# B&R Automation Studio project 305841_E00002_AM_0 (part 14)

#### ActionMotionFbs.st
```iecst
(********************************************************************
 * COPYRIGHT -- General Atomics
 ********************************************************************
 * Program: AxisStateMachine
 * File: ActionMoveVel.st
 * Author: Administrator
 * Created: January 22, 2014
 ********************************************************************
 * Implementation of program AxisStateMachine
 ********************************************************************)

ACTION ActionCallMotionFunctions:
  ActionMpAxisBasic;
  ActionCamInOut;
  ActionGearInOut;
  ActionOffsetShift;
  ActionPhaseShift;
END_ACTION

ACTION ActionMpAxisBasic:
  // 1) Range checks position, velocity, accel & Decel
  // 2) Packs the sMot_MoveParameters into a local axisBasicParamsStructure
  // 3) Detects parameter changes and manages the Update and UpdateDone bits
  // 4) Sets the fb command bits based on the axis sMot_AxisCommands structure
  // 5) Runs the fbMpAxisBasic funciton block
  // 6) Updates the axis structure with the status and axis info coming back from the fb

  // Make sure min/max values are not exceeded for position, velocity, accel, and decel.
  // Clamp if necessary

  // Position
  IF ax.MoveParameters.Position >  axPositionLimits.PositionLimitPos THEN
    ax.MoveParameters.Position :=  axPositionLimits.PositionLimitPos;
  END_IF;
  IF ax.MoveParameters.Position <  axPositionLimits.PositionLimitNeg THEN
    ax.MoveParameters.Position :=  axPositionLimits.PositionLimitNeg;
  END_IF;

  // Velocity
  IF ax.MoveParameters.Velocity > ax.MoveParameters.VelocityMax THEN
    ax.MoveParameters.Velocity := ax.MoveParameters.VelocityMax;
  END_IF;
  IF ax.MoveParameters.Velocity < ax.MoveParameters.VelocityMin THEN
    ax.MoveParameters.Velocity := ax.MoveParameters.VelocityMin;
  END_IF;

  // Accel and decel
  IF ax.MoveParameters.Acceleration > ax.MoveParameters.AccelMax THEN
    ax.MoveParameters.Acceleration := ax.MoveParameters.AccelMax;
  END_IF;
  IF ax.MoveParameters.Acceleration < ax.MoveParameters.AccelMin THEN
    ax.MoveParameters.Acceleration := ax.MoveParameters.AccelMin;
  END_IF;

  IF ax.MoveParameters.Deceleration > ax.MoveParameters.DecelMax THEN
    ax.MoveParameters.Deceleration := ax.MoveParameters.DecelMax;
  END_IF;
  IF ax.MoveParameters.Deceleration < ax.MoveParameters.DecelMin THEN
    ax.MoveParameters.Deceleration := ax.MoveParameters.DecelMin;
  END_IF;

  // The execution behavior is determined by the inputs set elsewhere
  // in particular the sMot_AxisCommands XxxxCmd bits,
  // and the values in sMot_MoveParameters structure

  // Axis reference set in init routine

  // Only enable the fb if the axis is not set to be ignored
  // TODO: Different check needed? Not sure how to tell if an axis reference is not set
  // It would be nice to check ax.fbMpAxisBasic.MpLink <> 0 for example, but this is a structure not an address
  IF NOT ax.Ignore AND ax.AxisNo <> 0 THEN
    ax.fbMpAxisBasic.Enable := TRUE;
  ELSE
    ax.fbMpAxisBasic.Enable := FALSE;
  END_IF;

  // Load the parameters from the sMot_MoveParameter structure into
  // local structure variables used for the fb
  fctPackMpAxisBasicParams(_I_UdtParams:= ADR(ax.MoveParameters), _IO_MpParams := axisBasicParams);

  // To allow move parameter changes to take effect without having to stop,
  // detect a difference between the desired parameters and the previous values.
  // If they are different, then set the update bit until the UpdateDone bit is set.
  // NOTE: This fb manages the ax.fbMpAxisCoupling.Update request and monitors the .UpdateDone bit
  // Use the .UpdateCouplingParams bit in the command structure if the application needs to control
  // when to trigger the update. If parameters need to be set in possibly different areas of the software,
  // and all the updates should take place at once, the update fb is called conditionally. The
  // checked bit can be set high so it is called all the time if the checked bit is not managed.
  ax.Commands.UpdateMoveParams:= TRUE;
  IF ax.Commands.UpdateMoveParams THEN
    ax.fbUpdateBFbParams(_IO_MpParams := axisBasicParams);
    ax.Commands.UpdateMoveParams := FALSE;
  END_IF;

  // TODO: Enforce move permissives

  // Use the commands from the axis structue
  ax.fbMpAxisBasic.ErrorReset := ax.Commands.DriveResetCmd;
  ax.fbMpAxisBasic.Power := ax.Commands.EnableCmd;
  ax.fbMpAxisBasic.Home := ax.Commands.HomeCmd;
  // There is no specific jog cmd. Use Move Velocity instead.
  ax.fbMpAxisBasic.MoveVelocity := ax.Commands.MoveVelocityCmd OR ax.Commands.MoveJogCmd;
  ax.fbMpAxisBasic.MoveAbsolute := ax.Commands.MoveAbsoluteCmd;
  ax.fbMpAxisBasic.MoveAdditive := ax.Commands.MoveRelativeCmd;
  ax.fbMpAxisBasic.Stop := ax.Commands.StopCmd;
  ax.fbMpAxisBasic.JogPositive := ax.Commands.MoveJogPositiveCmd;
  ax.fbMpAxisBasic.JogNegative := ax.Commands.MoveJogNegativeCmd;
  ax.fbMpAxisBasic.LimitLoad := ax.MoveParameters.EnableTorqueLimit;
  ax.fbMpAxisBasic.ReleaseBrake := ax.Commands.ReleaseBrakeCmd;
  ax.fbMpAxisBasic.AutoTune := FALSE; // TODO
  ax.fbMpAxisBasic.Simulate := FALSE; // TODO

  // Call the fb
  ax.fbMpAxisBasic();

  // Update the axis status structure
  ax.Status.Position := ax.fbMpAxisBasic.Position;
  ax.Status.Velocity := ax.fbMpAxisBasic.Velocity;
  ax.Status.IsPoweredOn := ax.fbMpAxisBasic.PowerOn;
  ax.Status.IsHomed := ax.fbMpAxisBasic.IsHomed;
  ax.Status.IsInVelocity := ax.fbMpAxisBasic.InVelocity;
  ax.Status.IsInPosition := ax.fbMpAxisBasic.InPosition;
  ax.Status.IsMoveActive := ax.fbMpAxisBasic.MoveActive;
  ax.Status.IsMoveDone := ax.fbMpAxisBasic.MoveDone;
  ax.Status.IsStopped := ax.fbMpAxisBasic.Stopped;
  ax.Status.IsTorqueLimitReady := ax.fbMpAxisBasic.LimitLoadReady;
  ax.Status.IsBrakeManuallyReleased := ax.fbMpAxisBasic.BrakeReleased;

  // Now load the sMot_AxisStatus structure with the data returned from the fb
  fctGetMpAxisInfo(_I_MpInfo := ADR(ax.fbMpAxisBasic.Info), _IO_UdtStatus := ax.Status);

  // Calculate special (algorithmic) positions
  CalcSpecialPositions;

  // Now that the status of this axis is known, copy it to the other axes slave status
  // area if this axis is specified as a slave.
  CopySlaveStatusToMaster;

END_ACTION

ACTION ActionCamInOut:
  // Execute the cam in or cam out fbs based on the CamIn/Out requests
  // The fbs are edge triggered, and the requests are cleared once serviced.
  // If the caming params change, another request must be made.
  // TODO: Is cam out and another cam in needed if params change?

  // Only execute the cam in fb if the axis number has been set,
  // the slave axis number has been set, and neither is set to be ignored,
  // and it is requested.
  IF ax.Ignore OR ax.AxisNo = AD_UNKNOWN OR
       ax.CouplingParameters.SlaveAxisNo = AD_UNKNOWN OR
       axes[ax.CouplingParameters.SlaveAxisNo].Ignore THEN
    // slave or master should be ignored
    // keep the requests and executes low
    ax.CouplingParameters.CamInReq := FALSE;
    ax.CouplingParameters.CamOutReq := FALSE;
    ax.fbCamIn.Execute := FALSE;
    ax.fbCamOut.Execute := FALSE;
  ELSIF ax.CouplingParameters.CamInReq THEN
    // CamIn request is made.
    // Clear the req so a future rising edge can be seen
    ax.CouplingParameters.CamInReq := FALSE;
    // Make sure the CamOut req and execute is clear
    ax.CouplingParameters.CamOutReq := FALSE;
    ax.fbCamOut.Execute := FALSE;
    // Load the cam in params, then set the execute input (edge triggered fb)
    ax.fbCamIn.MasterOffset := ax.CouplingParameters.CamMasterOffset;
    ax.fbCamIn.SlaveOffset := ax.CouplingParameters.CamSlaveOffset;
    ax.fbCamIn.MasterScaling := ax.CouplingParameters.CamScalingMaster;
    ax.fbCamIn.SlaveScaling := ax.CouplingParameters.CamScalingSlave;
    ax.fbCamIn.StartMode := ax.CouplingParameters.CamStartMode;
    ax.fbCamIn.MasterValueSource := ax.CouplingParameters.CamMasterValueSource;
    ax.fbCamIn.CamID := ax.CouplingParameters.CamId;
    ax.fbCamIn.BufferMode := ax.CouplingParameters.CamBufferMode; // only mcAborting currently supported
    ax.fbCamIn.AdvancedParameters.Periodic := ax.CouplingParameters.CamIsPeriodic;
    ax.fbCamIn.AdvancedParameters.Velocity := 0.0; // disable, use (slave?) axis max vel
    ax.fbCamIn.AdvancedParameters.Acceleration := 0.0; // disable, use (slave?) axis max accel
    ax.fbCamIn.AdvancedParameters.Deceleration := 0.0; // disable, use (slave?) axis max decel
    ax.fbCamIn.AdvancedParameters.Jerk := 0.0; // only non-zero if using McProfGen
    ax.fbCamIn.Execute := TRUE; // fb looks for a rising edge
  ELSIF ax.CouplingParameters.CamOutReq THEN
    // Clear the req so a future rising edge can be seen
    ax.CouplingParameters.CamOutReq := FALSE;
    // Make sure the GearIn req and execute is clear
    ax.CouplingParameters.CamInReq := FALSE;
    ax.fbCamIn.Execute := FALSE;
    // Load the cam out params, then set the execute input (edge triggered fb)
    ax.fbCamOut.Jerk := 0.0; // only non-zero if using McProfGen
    ax.fbCamOut.Execute := TRUE;
  END_IF;

  // Call the cam in and cam out fbs.
  ax.fbCamIn();
  ax.fbCamOut();
  // Clear the exuecute bits. The fbs are edge triggerd, and would have been seen by the above call.
  ax.fbCamIn.Execute := FALSE;
  ax.fbCamOut.Execute := FALSE;

  // Update the axis status structure
  IF ax.fbCamIn.Active AND NOT ax.fbCamIn.Error THEN
    ax.Status.IsCamInSync := ax.fbCamIn.InSync;
    ax.Status.IsCamEndOfProfile := ax.fbCamIn.EndOfProfile;
    ax.Status.CamStatus := ax.fbCamIn.Status;
  ELSE
    ax.Status.IsCamInSync := FALSE;
    ax.Status.IsCamEndOfProfile := FALSE;
    ax.Status.CamStatus := mcCAM_STATUS_PREPARING_MOVE; // 0 value, but don't have a good choice for "not active
  END_IF;

END_ACTION

ACTION ActionGearInOut:
  // Execute the gear in or gear out fbs based on the GearIn/Out requests
  // The fbs are edge triggered, and the requests are cleared once serviced.
  // If the gearing params change, another request must be made.

  // Only execute the gear in fb if the axis number has been set,
  // the slave axis number has been set, and neither is set to be ignored,
  // and it is requested.
  IF ax.Ignore OR ax.AxisNo = AD_UNKNOWN OR
       ax.CouplingParameters.SlaveAxisNo = AD_UNKNOWN OR
       axes[ax.CouplingParameters.SlaveAxisNo].Ignore THEN
    // slave or master should be ignored
    // keep the requests and executes low
    ax.CouplingParameters.GearInReq := FALSE;
    ax.CouplingParameters.GearOutReq := FALSE;
    ax.fbGearIn.Execute := FALSE;
    ax.fbGearOut.Execute := FALSE;
  ELSIF ax.CouplingParameters.GearInReq THEN
    // GearIn request is made.
    // Clear the req so a future rising edge can be seen
    ax.CouplingParameters.GearInReq := FALSE;
    // Make sure the GearOut req and execute is clear
    ax.CouplingParameters.GearOutReq := FALSE;
    ax.fbGearOut.Execute := FALSE;
    // Load the gear in params, then set the execute input (edge triggered fb)
    ax.fbGearIn.RatioNumerator := ax.CouplingParameters.GearInRatioNumerator;
    ax.fbGearIn.RatioDenominator := ax.CouplingParameters.GearInRatioDenominator;
    ax.fbGearIn.MasterValueSource := ax.CouplingParameters.GearInMasterValueSource;
    ax.fbGearIn.Acceleration := ax.CouplingParameters.ShiftAccelerationMax;
    ax.fbGearIn.Deceleration := ax.CouplingParameters.ShiftDecelerationMax;
    ax.fbGearIn.Jerk := ax.CouplingParameters.ShiftJerk; // only non-zero if using McProfGen
    ax.fbGearIn.BufferMode := ax.CouplingParameters.GearInBufferMode; // onlly mcAborting currently supported
    ax.fbGearIn.AdvancedParameters.MasterMaxVelocity := ax.CouplingParameters.ShiftProfileBaseMaxVelocity;
    ax.fbGearIn.Execute := TRUE; // fb looks for a rising edge
  ELSIF ax.CouplingParameters.GearOutReq THEN
    // Clear the req so a future rising edge can be seen
    ax.CouplingParameters.GearOutReq := FALSE;
    // Make sure the GearIn req and execute is clear
    ax.CouplingParameters.GearInReq := FALSE;
    ax.fbGearIn.Execute := FALSE;
    // Load the gear out params, then set the execute input (edge triggered fb)
    ax.fbGearOut.Jerk := 0.0; // only non-zero if using McProfGen
    ax.fbGearOut.Execute := TRUE;
  END_IF;

  // Call the gear in and gear out fbs.
  ax.fbGearIn();
  ax.fbGearOut();
  // Clear the exuecute bits. The fbs are edge triggerd, and would have been seen by the above call.
  ax.fbGearIn.Execute := FALSE;
  ax.fbGearOut.Execute := FALSE;

  // Update the axis status structure.
  // Derrive InCompensation -- Active but not in sync
  IF ax.fbGearIn.Active AND NOT ax.fbGearIn.Error THEN
    // If gear in is active, it is either in sync or in compensation
    ax.Status.IsGearInSync := ax.fbGearIn.InGear;
    ax.Status.IsGearInCompensation := NOT ax.fbGearIn.InGear;
  ELSE
    ax.Status.IsGearInSync := FALSE;
    ax.Status.IsGearInCompensation := FALSE;
  END_IF;

END_ACTION

ACTION ActionOffsetShift:
  // Execute the offset shift fb based on the offset shift request.
  // The fb is edge triggered, and the request is cleared once serviced.
  // If the offset params change, another request must be made.

  // Only execute the offset shift fb if the axis number has been set,
  // the slave axis number has been set, and neither is set to be ignored,
  // and it is requested.
  IF ax.Ignore OR ax.AxisNo = AD_UNKNOWN OR
       ax.CouplingParameters.SlaveAxisNo = AD_UNKNOWN OR
       axes[ax.CouplingParameters.SlaveAxisNo].Ignore THEN
    // slave or master should be ignored
    // keep the request and enable low
    ax.CouplingParameters.OffsetShiftReq := FALSE;
    ax.fbOffsetShift.Enable := FALSE;
    ax.fbOffsetShift.StartShift := FALSE;
  ELSE
    ax.fbOffsetShift.Enable := TRUE;
  END_IF;

  // Enable input and ignore considered above. If req is high,
  // it can be acted upon.
  IF ax.CouplingParameters.OffsetShiftReq THEN
    // Offset Shift request is made.
    // Clear the req so a future rising edge can be seen
    ax.CouplingParameters.OffsetShiftReq := FALSE;
    // Load the offset shift params, then set the start shift input (edge sensitive input)
    ax.fbOffsetShift.OffsetShift := ax.CouplingParameters.Shift;
    ax.fbOffsetShift.Velocity := ax.CouplingParameters.ShiftVelocityMax;
    ax.fbOffsetShift.Acceleration := ax.CouplingParameters.ShiftAccelerationMax;
    ax.fbOffsetShift.AdvancedParameters.ShiftMode := ax.CouplingParameters.ShiftMode;
    ax.fbOffsetShift.AdvancedParameters.ProfileBase := ax.CouplingParameters.ShiftProfileBase;
    ax.fbOffsetShift.AdvancedParameters.ProfileBaseMaxVelocity := ax.CouplingParameters.ShiftProfileBaseMaxVelocity;
    ax.fbOffsetShift.AdvancedParameters.DistanceParameters.ProfileDistance := ax.CouplingParameters.ShiftProfileDistance;
    ax.fbOffsetShift.AdvancedParameters.ZoneParameters.StartPosition := ax.CouplingParameters.ShiftZoneStartPosition;
    ax.fbOffsetShift.AdvancedParameters.ZoneParameters.EndPosition := ax.CouplingParameters.ShiftZoneEndPosition;
    ax.fbOffsetShift.AdvancedParameters.ZoneParameters.Period := ax.CouplingParameters.ShiftZonePeriod;
    ax.fbOffsetShift.AdvancedParameters.ShiftAlternativeValueSource := mcALT_VALUE_NOT_USED;
    ax.fbOffsetShift.StartShift := TRUE; // fb looks for a rising edge
  END_IF;

  // Call the offset shift fb.
  ax.fbOffsetShift();
  // Clear the start shift bit. The fb is edge triggerd, and it would have been seen by the above call.
  ax.fbOffsetShift.StartShift := FALSE; // fb looks for a rising edge

  // Update the axis status structure as long as status is valid and there is no error.
  // Otherwise, clear the values
  IF ax.fbOffsetShift.Valid AND NOT ax.fbOffsetShift.Error THEN
    ax.Status.IsCoordOffsetShiftAttained := ax.fbOffsetShift.ShiftAttained;
    ax.Status.IsCoordOffsetShiftStarted := ax.fbOffsetShift.ShiftStarted;
    ax.Status.CoordActualOffsetShift := ax.fbOffsetShift.ActualOffsetShift;
  ELSE
    ax.Status.IsCoordOffsetShiftAttained := FALSE;
    ax.Status.IsCoordOffsetShiftStarted := FALSE;
    ax.Status.CoordActualOffsetShift := 0.0;
  END_IF;

END_ACTION

ACTION ActionPhaseShift:
  // Execute the phase shift fb based on the phase shift request.
  // The fb is edge triggered, and the request is cleared once serviced.
  // If the phase params change, another request must be made.
  // TODO: Verify operation/behavior when changing params

  // Only execute the phase shift fb if the axis number has been set,
  // the slave axis number has been set, and neither is set to be ignored,
  // and it is requested.
  IF ax.Ignore OR ax.AxisNo = AD_UNKNOWN OR
       ax.CouplingParameters.SlaveAxisNo = AD_UNKNOWN OR
       axes[ax.CouplingParameters.SlaveAxisNo].Ignore THEN
    // slave or master should be ignored
    // keep the request and enable low
    ax.CouplingParameters.PhaseShiftReq := FALSE;
    ax.fbPhaseShift.Enable := FALSE;
    ax.fbPhaseShift.StartShift := FALSE;
  ELSE
    ax.fbPhaseShift.Enable := TRUE;
  END_IF;

  // Enable input and ignore considered above. If req is high,
  // it can be acted upon.
  IF ax.CouplingParameters.PhaseShiftReq THEN
    // Phase Shift request is made.
    // Clear the req so a future rising edge can be seen
    ax.CouplingParameters.PhaseShiftReq := FALSE;
    // Load the phase shift params, then set the start shift input (edge sensitive input)
    ax.fbPhaseShift.PhaseShift := ax.CouplingParameters.Shift;
    ax.fbPhaseShift.Velocity := ax.CouplingParameters.ShiftVelocityMax;
    ax.fbOffsetShift.Acceleration := ax.CouplingParameters.ShiftAccelerationMax;
    ax.fbOffsetShift.AdvancedParameters.ShiftMode := ax.CouplingParameters.ShiftMode;
    ax.fbOffsetShift.AdvancedParameters.ProfileBase := ax.CouplingParameters.ShiftProfileBase;
    ax.fbOffsetShift.AdvancedParameters.ProfileBaseMaxVelocity := ax.CouplingParameters.ShiftProfileBaseMaxVelocity;
    ax.fbOffsetShift.AdvancedParameters.DistanceParameters.ProfileDistance := ax.CouplingParameters.ShiftProfileDistance;
    ax.fbOffsetShift.AdvancedParameters.ZoneParameters.StartPosition := ax.CouplingParameters.ShiftZoneStartPosition;
    ax.fbOffsetShift.AdvancedParameters.ZoneParameters.EndPosition := ax.CouplingParameters.ShiftZoneEndPosition;
    ax.fbOffsetShift.AdvancedParameters.ZoneParameters.Period := ax.CouplingParameters.ShiftZonePeriod;
    ax.fbOffsetShift.AdvancedParameters.ShiftAlternativeValueSource := mcALT_VALUE_NOT_USED;
    ax.fbPhaseShift.StartShift := TRUE; // fb looks for a rising edge
  END_IF;

  // Call the phase shift fb.
  ax.fbPhaseShift();
  // Clear the start shift bit. The fb is edge triggerd, and it would have been seen by the above call.
  ax.fbPhaseShift.StartShift := FALSE; // fb looks for a rising edge

  // Update the axis status structure as long as status is valid and there is no error.
  // Otherwise, clear the values
  IF ax.fbPhaseShift.Valid AND NOT ax.fbPhaseShift.Error THEN
    ax.Status.IsCoordPhaseShiftAttained := ax.fbPhaseShift.ShiftAttained;
    ax.Status.IsCoordPhaseShiftStarted := ax.fbPhaseShift.ShiftStarted;
    ax.Status.CoordActualPhaseShift := ax.fbPhaseShift.ActualPhaseShift;
  ELSE
    ax.Status.IsCoordPhaseShiftAttained := FALSE;
    ax.Status.IsCoordPhaseShiftStarted := FALSE;
    ax.Status.CoordActualPhaseShift := 0.0;
  END_IF;

END_ACTION

ACTION CopySlaveStatusToMaster :
  // If this axis number is a slave to another axis, then copy this axis
  // status to the master axis structure. This is a convenience
  // so the HMI for example, only needs to look in one structure (the master) and
  // can access the slave status.

  // Loop thru the axes. If the axis of index has this axis specified as a slave axis,
  // copy this axis status to the axis of index slave status.
  // Axis 0 is a dummy axis, so it can be skipped.
  FOR axIdx := 1 TO AXIS_COUNT DO
    IF axes[axIdx].CouplingParameters.SlaveAxisNo = AXIS_NO THEN
      // This axis is a slave to the axis referenced by axIdx.
      // Copy this axis status to the indexed axis slave status
      fctCopyAxisStatus(_I_SrcStatus := ADR(ax.Status), _I_DestStatus := ADR(axes[axIdx].StatusSlave));
    END_IF;
  END_FOR;
END_ACTION
```

- ActionMotionFbs.st.bak (not shown)

#### AxSMInit.st
```iecst
PROGRAM _INIT
  // set ax pointer to the element of the global sMot_Axis array
  ax ACCESS ADR(axes[AXIS_NO]);

  // set the position limits to point to the global permanent variable
  axPositionLimits ACCESS ADR(gr_AxisPositionLimits[AXIS_NO]);

  // Set the axis number and clear the ignore bit
  ax.AxisNo:= AXIS_NO;

  // **** These settings need to be reviewed/set for each axis
  ax.CouplingParameters.SlaveAxisNo := DINT_TO_USINT(AD_UNKNOWN); // This axis will have slaves, but it changes during run-time
  ax.Ignore := FALSE;
  ax.isAxisEndless := TRUE;
  ax.isAxisVirtual := TRUE;
  ax.isAxisInverter := FALSE;

  // Point to the mappMotion axis, and a slave if there is one
  ax.AxisObj := gvAxHw; // mappMotion axis -- see mappMotion in cfg view
  ax.SlaveAxisObj := axDummySlave; // slave axis for the handwheel is dynamic

  // Set the restore pos check fb
  // ax.fbCheckRestorePos.Axis := ADR(ax.AxisObj);
  // ax.fbCheckRestorePos.DataAddress := ADR(gr_AxHwRestorePos); // Set this per axis

  // Load the min/max velocity and accel/decel from constants
  // Note: Moves not used for virtual axes, so values are not important
  ax.MoveParameters.AccelMin := 0.001; // TODO: Not sure of a good value, but it should not be zero.
  ax.MoveParameters.AccelMax:= 10.0;
  ax.MoveParameters.DecelMin := 0.001; // TODO:Not sure of a good value, but it should not be zero.
  ax.MoveParameters.DecelMax:= 10.0;
  ax.MoveParameters.VelocityMin := 0.000;
  ax.MoveParameters.VelocityMax := 01.0;

  // **** The settings below don't normally need to be altered

  // set the fb axis references
  ax.fbMpAxisBasic.MpLink := ADR(ax.AxisObj);
  ax.fbReadDrivePos.Axis:= ADR(ax.AxisObj);
  ax.fbGearIn.Master := ADR(ax.AxisObj);
  ax.fbGearIn.Slave := ADR(ax.SlaveAxisObj);
  ax.fbGearOut.Slave := ADR(ax.SlaveAxisObj);
  ax.fbOffsetShift.Slave := ADR(ax.SlaveAxisObj);
  ax.fbPhaseShift.Slave := ADR(ax.SlaveAxisObj);
  ax.fbCamIn.Master := ADR(ax.AxisObj);
  ax.fbCamIn.Slave := ADR(ax.SlaveAxisObj);
  ax.fbCamOut.Slave := ADR(ax.SlaveAxisObj);
  ax.fbUpdateBFbParams._I_Axis := ADR(ax);

  // Set fb reference to local variables
  ax.fbMpAxisBasic.Parameters := ADR(axisBasicParams);

  // Set previous values for motion parameters so changes can be detected
  ax.MoveParametersPrev := ax.MoveParameters;

  // Clear commands and requests
  fctClearMotionCommands(_I_CmdMask := MACM_NOMASK, _IO_Commands := ax.Commands);
  fctClearMotionRequests(_I_ReqMask := MACM_NOMASK, _IO_Commands := ax.Commands);

  // set the move not allowed flag
  ax.Commands.MoveNotAllowed:= TRUE;

  // Set the most primitive status. If the axis is valid, the
  // full status will be updated later once comms is established, and the drive status is updated via MpAxisBasic
  ax.Status.IsCommuncationReady := FALSE;
  ax.Status.IsReadyToPowerOn := FALSE;

END_PROGRAM
```

### Program Logical/PlcLogic/axCfVfd/axCfVfdSM

#### AxSM.var
```iecst
(********************************************************************
 * COPYRIGHT -- General Atomics
 ********************************************************************
 * Program: AFtInSM
 * File: AFtInSM.var
 * Author: Administrator
 * Created: July 16, 2014
 ********************************************************************
 * Local variables of program AFtInSM
 ********************************************************************)
VAR CONSTANT
  (* axis number is per eAXIS_DESIGNATION *)
  (*
    AD_UNKNOWN := 0,
    AD_SPINDLE := 1,
    AD_OUTER_ECCENTRIC := 2,
    AD_INNER_ECCENTRIC := 3,
    AD_Z := 4,
    derrived axes
    AD_X := 5,
    AD_Y := 6,
    virual axes
    AD_HANDWHEEL := 7
    AD_CF_VFD := 8
  *)

  (* same info but different data types for convenience *)
  AXIS_NO : USINT := AD_CF_VFD; (* USINT so it can be used as an array index *)
  AXIS_DESIGNATION : eAXIS_DESIGNATION := AD_CF_VFD;

  END_VAR

  VAR
  ax : REFERENCE TO sMot_Axis;
  axPositionLimits : REFERENCE TO sMot_PositionLimits;
  axIdx : DINT; (* axis index *)
  axDummySlave : McAxisType;
	(* local versions of motion param structures -- used to make setting advanced params easier *)
  axisBasicParams : MpAxisBasicParType;
  tmrStepTO : TON; (* Step TO timer *)
  reqMask : DINT := MACM_NOMASK; (* request mask *)
  cmdMask : DINT := MACM_NOMASK; (* command mask *)
  tmrDriveReset : TON; (* auto issue drive reset while invalid also used to force minimum time in error states *)
	tmrModeMismatch : TON; (* mode mismatch timer *)
	tmrHomeMinimum : TON; (* force Home cmd to be present before transitioning *)
END_VAR
```

#### ActionChkPermissives.st
```iecst
(********************************************************************
 * COPYRIGHT -- General Atomics
 ********************************************************************
 * Program: AxisStateMachine
 * File: ActionCheckPermissiveJog.st
 * Author: Administrator
 * Created: June 02, 2014
 ********************************************************************
 * Implementation of program AxisStateMachine
 ********************************************************************)

ACTION ActionChkPermissiveContinuous:
  // Permissive check for continuous moves -- jogs and velocity
  // These moves have an undefined length

  // NOTE THE MOVE NOT ALLOWED FLAG: This aciton will set this flag if it finds the move to be in violation.
  // It does not clear the flag, however, and this allows several check actions to be called in a chain. If
  // at the end of all the calls, the flag is set, then it is intended that the overall application logic should
  // not allow the move.

  (* ***** WARNING CAUTION ****
  These checks have only primitive checks for taking into account current velocicy, deceleration, and stopping distance.
  This means that the permissives will try to honor position limits, and try to keep from over-running a limit,
  but may overshoot if you run right up to a limit.

  The stopping distance is calculated from the velocity and decel value, which is mathmatically correct, but
  in practice, the velocity value is approximate since it is sampled at a relatively slow rate.
  ***************************** *)

  // Calculate the stopping Distance if the axis is not virtual
  // If the axis in not moving, assume the velocity parameter for a move.
  // If the axis is moving, used the reported velocity
  // Stopping distance = Vavg * t => V/2 * V/decel => V^2/2*decel
  IF NOT ax.isAxisVirtual THEN
    IF  ax.Status.PlcOpenState = mcAXIS_CONTINUOUS_MOTION OR // Will probably be continuous or synchronized because
        ax.Status.PlcOpenState = mcAXIS_DISCRETE_MOTION OR
        ax.Status.PlcOpenState = mcAXIS_SYNCHRONIZED_MOTION THEN
      // Axis is moving ... Use reported velocity
      // Prevent against divide by zero by assuming a value if decel is zero
      IF ax.MoveParameters.Deceleration = 0.0 THEN
        // No valid decel. Use min decel
        ax.MoveParameters.PermissiveCheck.EstStoppingDistance := (ax.Status.Velocity ** 2) / (2.0 * ax.MoveParameters.DecelMin);
      ELSE
        // We have a decel value, so use that
        ax.MoveParameters.PermissiveCheck.EstStoppingDistance := (ax.Status.Velocity ** 2) / (2.0 * ax.MoveParameters.Deceleration);
      END_IF;
    ELSE
      // Axis is stopped ... assume parameter velocity
      // Prevent against divide by zero by assuming a small value if decel is zero
      IF ax.MoveParameters.Deceleration = 0.0 THEN
        // No valid decel. Use min decel.
        ax.MoveParameters.PermissiveCheck.EstStoppingDistance := (ax.MoveParameters.Velocity ** 2) / (2.0 * ax.MoveParameters.DecelMin);
      ELSE
        // We have a decel value, so use that
        ax.MoveParameters.PermissiveCheck.EstStoppingDistance := (ax.MoveParameters.Velocity ** 2) / (2.0 * ax.MoveParameters.Deceleration);
      END_IF;
    END_IF;
  ELSE
    // virtual axis does not allow moves, so done not need stopping distance.
    ax.MoveParameters.PermissiveCheck.EstStoppingDistance := 0.0;
  END_IF;

  // Check the directional move permissives and then check the allowable position range

  // Initially clear the Check Failed flag.
  // This will get set if any check fails.
  // It will get checked at the end and will get used to control the
  // move not allowed bit. The move not allowed bit was not used directly in the
  // intermediate checks to avoid it transiting until all the logic was complete
  ax.MoveParameters.PermissiveCheck.CheckFailed:= FALSE;

  // positive move permissive
  IF ax.MoveParameters.Direction = mcDIR_POSITIVE  AND NOT ax.MoveParameters.PosMovePermissive THEN
    ax.MoveParameters.PermissiveCheck.PermissiveHaltPos:= TRUE;
    ax.MoveParameters.PermissiveCheck.CheckFailed:= TRUE;
  ELSE
    ax.MoveParameters.PermissiveCheck.PermissiveHaltPos:= FALSE;
  END_IF;

  // negative move permissive
  IF ax.MoveParameters.Direction = mcDIR_NEGATIVE AND NOT ax.MoveParameters.NegMovePermissive THEN
    ax.MoveParameters.PermissiveCheck.PermissiveHaltNeg:= TRUE;
    ax.MoveParameters.PermissiveCheck.CheckFailed:= TRUE;
  ELSE
    ax.MoveParameters.PermissiveCheck.PermissiveHaltNeg:= FALSE;
  END_IF;

  // If the check passed the above, and the axis is not endless, then check the position limits
  IF NOT ax.MoveParameters.PermissiveCheck.CheckFailed AND NOT ax.isAxisEndless THEN
    // positive position window
    IF ax.MoveParameters.Direction = mcDIR_POSITIVE  AND
      (ax.Status.Position >=  axPositionLimits.PositionLimitPos OR
      ax.Status.Position + ax.MoveParameters.PermissiveCheck.EstStoppingDistance >=  axPositionLimits.PositionLimitPos) THEN
      ax.MoveParameters.PermissiveCheck.RangeLimitPos:= TRUE;
      ax.MoveParameters.PermissiveCheck.CheckFailed:= TRUE;
    ELSE
      ax.MoveParameters.PermissiveCheck.RangeLimitPos:= FALSE;
    END_IF;

    // negative position window
    IF ax.MoveParameters.Direction = mcDIR_NEGATIVE AND
      (ax.Status.Position <=  axPositionLimits.PositionLimitNeg OR
      ax.Status.Position - ax.MoveParameters.PermissiveCheck.EstStoppingDistance <=  axPositionLimits.PositionLimitNeg) THEN
      ax.MoveParameters.PermissiveCheck.RangeLimitNeg:= TRUE;
      ax.MoveParameters.PermissiveCheck.CheckFailed:= TRUE;
    ELSE
      ax.MoveParameters.PermissiveCheck.RangeLimitNeg:= FALSE;
    END_IF;
  ELSIF ax.isAxisEndless THEN
    // Axis is endless, so it won't fail on position range... clear the bits
    ax.MoveParameters.PermissiveCheck.RangeLimitPos := FALSE;
    ax.MoveParameters.PermissiveCheck.RangeLimitNeg := FALSE;
  END_IF;

  // Set move not allowed bit depending on the check failed flag
  IF ax.MoveParameters.PermissiveCheck.CheckFailed THEN
    // at least 1 permissive failed, don't allow the move
    ax.Commands.MoveNotAllowed:= TRUE;
  END_IF;

END_ACTION

ACTION ActionChkPermissiveRel:
  // Check the directional move permissives and then check the allowable position range

  // NOTE THE MOVE NOT ALLOWED FLAG: This aciton will set this flag if it finds the move to be in violation.
  // It does not clear the flag, however, and this allows several check actions to be called in a chain. If
  // at the end of all the calls, the flag is set, then it is intended that the overall application logic should
  // not allow the move.

  // Initially clear the Check Failed flag.
  // This will get set if any check fails.
  // It will get checked at the end and will get used to control the
  // move not allowed bit. The move not allowed bit was not used directly in the
  // intermediate checks to avoid it transiting until all the logic was complete
  ax.MoveParameters.PermissiveCheck.CheckFailed:= FALSE;

  // positive move permissive
  // if distance is > 0, move is positive
  IF ax.MoveParameters.Distance > 0 AND NOT ax.MoveParameters.PosMovePermissive THEN
    ax.MoveParameters.PermissiveCheck.PermissiveHaltPos:= TRUE;
    ax.MoveParameters.PermissiveCheck.CheckFailed:= TRUE;
  ELSE
    ax.MoveParameters.PermissiveCheck.PermissiveHaltPos:= FALSE;
  END_IF;

  // negative move permissive
  // if distance is < 0, move is negative
  IF ax.MoveParameters.Distance < 0 AND NOT ax.MoveParameters.NegMovePermissive THEN
    ax.MoveParameters.PermissiveCheck.PermissiveHaltNeg:= TRUE;
    ax.MoveParameters.PermissiveCheck.CheckFailed:= TRUE;
  ELSE
    ax.MoveParameters.PermissiveCheck.PermissiveHaltNeg:= FALSE;
  END_IF;

  // If the check passed the above, and the axis is not endless, then check the position limits
  IF NOT ax.MoveParameters.PermissiveCheck.CheckFailed AND NOT ax.isAxisEndless THEN
    // positive position window -- if distance is > 0, move is positive
    IF ax.MoveParameters.Distance > 0.0 AND
      ax.MoveParameters.PermissiveCheck.StartPosition + ax.MoveParameters.Distance > axPositionLimits.PositionLimitPos THEN
      ax.MoveParameters.PermissiveCheck.RangeLimitPos:= TRUE;
      ax.MoveParameters.PermissiveCheck.CheckFailed:= TRUE;
    ELSE
      ax.MoveParameters.PermissiveCheck.RangeLimitPos:= FALSE;
    END_IF;

    // negative position window -- if distance is < 0, move is negative
    IF ax.MoveParameters.Distance < 0.0 AND
      ax.MoveParameters.PermissiveCheck.StartPosition + ax.MoveParameters.Distance < axPositionLimits.PositionLimitNeg THEN
      ax.MoveParameters.PermissiveCheck.RangeLimitNeg:= TRUE;
      ax.MoveParameters.PermissiveCheck.CheckFailed:= TRUE;
    ELSE
      ax.MoveParameters.PermissiveCheck.RangeLimitNeg:= FALSE;
    END_IF;
  ELSIF ax.isAxisEndless THEN
    // Axis is endless, so it won't fail on position range... clear the bits
    ax.MoveParameters.PermissiveCheck.RangeLimitPos := FALSE;
    ax.MoveParameters.PermissiveCheck.RangeLimitNeg := FALSE;
  END_IF;

  // Set the move not allowed bit depending on the check failed flag
  IF ax.MoveParameters.PermissiveCheck.CheckFailed THEN;
    // at least 1 permissive failed, don't allow the move
    ax.Commands.MoveNotAllowed:= TRUE;
  END_IF;

END_ACTION

ACTION ActionChkPermissiveAbs:
  // Check the directional move permissives and then check the allowable position range

  // NOTE THE MOVE NOT ALLOWED FLAG: This aciton will set this flag if it finds the move to be in violation.
  // It does not clear the flag, however, and this allows several check actions to be called in a chain. If
  // at the end of all the calls, the flag is set, then it is intended that the overall application logic should
  // not allow the move.

  // Initially clear the Check Failed flag.
  // This will get set if any check fails.
  // It will get checked at the end and will get used to control the
  // move not allowed bit. The move not allowed bit was not used directly in the
  // intermediate checks to avoid it transiting until all the logic was complete
  ax.MoveParameters.PermissiveCheck.CheckFailed:= FALSE;

  // Positive move permissive
  // If requested position is > than current position, the move is positive
  IF ax.MoveParameters.Position > ax.Status.Position AND NOT ax.MoveParameters.PosMovePermissive THEN
    ax.MoveParameters.PermissiveCheck.PermissiveHaltPos:= TRUE;
    ax.MoveParameters.PermissiveCheck.CheckFailed:= TRUE;
  ELSE
    ax.MoveParameters.PermissiveCheck.PermissiveHaltPos:= FALSE;
  END_IF;

  // Negative move permissive
  // If requested position is < than current position, the move is negative
  IF ax.MoveParameters.Position < ax.Status.Position AND NOT ax.MoveParameters.NegMovePermissive THEN
    ax.MoveParameters.PermissiveCheck.PermissiveHaltNeg:= TRUE;
    ax.MoveParameters.PermissiveCheck.CheckFailed:= TRUE;
  ELSE
    ax.MoveParameters.PermissiveCheck.PermissiveHaltNeg:= FALSE;
  END_IF;

  // If the check passed the above, and the axis is not endless, then check the position limits
  IF NOT ax.MoveParameters.PermissiveCheck.CheckFailed AND NOT ax.isAxisEndless THEN

    // Check that the requested position is within the allowable range
    // Positive position window
    IF ax.MoveParameters.Position >  axPositionLimits.PositionLimitPos THEN
      ax.MoveParameters.PermissiveCheck.RangeLimitPos:= TRUE;
      ax.MoveParameters.PermissiveCheck.CheckFailed:= TRUE;
    ELSE
      ax.MoveParameters.PermissiveCheck.RangeLimitPos:= FALSE;
    END_IF;

    // Negative position window
    IF ax.MoveParameters.Position <  axPositionLimits.PositionLimitNeg THEN
      ax.MoveParameters.PermissiveCheck.RangeLimitNeg:= TRUE;
      ax.MoveParameters.PermissiveCheck.CheckFailed:= TRUE;
    ELSE
      ax.MoveParameters.PermissiveCheck.RangeLimitNeg:= FALSE;
    END_IF;

  ELSIF ax.isAxisEndless THEN
    // Axis is endless, so it won't fail on position range... clear the bits
    ax.MoveParameters.PermissiveCheck.RangeLimitPos := FALSE;
    ax.MoveParameters.PermissiveCheck.RangeLimitNeg := FALSE;
  END_IF;

  // Set the move not allowed bit depending on the check failed flag
  IF ax.MoveParameters.PermissiveCheck.CheckFailed THEN;
    // at least 1 permissive failed, don't allow the move
    ax.Commands.MoveNotAllowed:= TRUE;
  END_IF;

END_ACTION

ACTION ActionChkPermissiveCoupling:
  // This action will consider the coupling status and determine if a move should be stopped.
  // If there is no coupled slave, this action won't set the move not allowed flag.
  // If there is a coupled slave, this action will stop the master if the slave stops.

  // NOTE THE MOVE NOT ALLOWED FLAG: This aciton will set this flag if it finds the move to be in violation.
  // It does not clear the flag, however, and this allows several check actions to be called in a chain. If
  // at the end of all the calls, the flag is set, then it is intended that the overall application logic should
  // not allow the move.

  // Initially clear the Check Failed flag.
  // This will get set if any check fails.
  // It will get checked at the end and will get used to control the
  // move not allowed bit. The move not allowed bit was not used directly in the
  // intermediate checks to avoid it transiting until all the logic was complete
  ax.MoveParameters.PermissiveCheck.CheckFailed:= FALSE;

  // Make sure to stop the master if the slave goes out of sync w/o being commanded to
  IF (ax.fbGearIn.Active OR ax.fbCamIn.Active) AND ax.StatusSlave.PlcOpenState = mcAXIS_SYNCHRONIZED_MOTION THEN
    // Slave is geared or cammed (in synchronized motion) Set the flag so loss of sync can be acted on
    // This flag gets cleared if GearOut or CamOut go active, or
    // if the master enteres the stopping, homing, disabled, or error stop state.
    ax.Status.HasCoordinatedSlave := TRUE;
  ELSIF (ax.fbGearOut.Done OR ax.fbCamOut.Done) OR
          // ax.Status.PlcOpenState = mcAXIS_STOPPING OR
          ax.Status.PlcOpenState = mcAXIS_HOMING OR
          ax.Status.PlcOpenState = mcAXIS_DISABLED OR
          ax.Status.PlcOpenState = mcAXIS_ERRORSTOP THEN
    // Slave is not geared or cammed. Clear the flag
    ax.Status.HasCoordinatedSlave := FALSE;
  END_IF;

  // If slave was synched or in compensation, and is still supposed to be synched (but isnt'), and the master is moving, then
  // stop the master.
  IF ax.Status.HasCoordinatedSlave AND ax.StatusSlave.PlcOpenState <> mcAXIS_SYNCHRONIZED_MOTION THEN
    // ax.MoveParameters.PermissiveCheck.CheckFailed:= TRUE;
    ax.Commands.HaltReq := TRUE;

  END_IF;

  // TODO: Are there other checks??
  // Not sure how to check an engaged slave because it does not know what the master will do.
  // Investigate what is needed. For now, allow the move. I think a real solution would need
  // to be based on the direction and distances for the master axis, and calculated thru a gear
  // ratio or cam to what the slave would do.

  // Set the move not allowed bit depending on the check failed flag
  IF ax.MoveParameters.PermissiveCheck.CheckFailed THEN;
    // at least 1 permissive failed, don't allow the move
    ax.Commands.MoveNotAllowed:= TRUE;
  END_IF;

  // The slave allows itself to be coupled by setting the coupling permissive in its own axis structure.
  // Allow coupling if homed, and in standstill (powered), discrete or continuous motion,
  // Or if it is already coupled
  ax.CouplingParameters.CouplingPermissive :=
    ax.Status.IsHomed AND
    (ax.Status.PlcOpenState = mcAXIS_STANDSTILL OR
     ax.Status.PlcOpenState = mcAXIS_DISCRETE_MOTION OR
     ax.Status.PlcOpenState = mcAXIS_CONTINUOUS_MOTION OR
     ax.Status.PlcOpenState = mcAXIS_SYNCHRONIZED_MOTION);

END_ACTION
```

#### ActionMotionFbs.st
```iecst
(********************************************************************
 * COPYRIGHT -- General Atomics
 ********************************************************************
 * Program: AxisStateMachine
 * File: ActionMoveVel.st
 * Author: Administrator
 * Created: January 22, 2014
 ********************************************************************
 * Implementation of program AxisStateMachine
 ********************************************************************)

ACTION ActionCallMotionFunctions:
  ActionMpAxisBasic;
  ActionMpAxisCoupling;
END_ACTION

ACTION ActionMpAxisBasic:
  // 1) Range checks position, velocity, accel & Decel
  // 2) Packs the sMot_MoveParameters into a local axisBasicParamsStructure
  // 3) Detects parameter changes and manages the Update and UpdateDone bits
  // 4) Sets the fb command bits based on the axis sMot_AxisCommands structure
  // 5) Runs the fbMpAxisBasic funciton block
  // 6) Updates the axis structure with the status and axis info coming back from the fb

  // Make sure min/max values are not exceeded for position, velocity, accel, and decel.
  // Clamp if necessary

  // Position
  IF ax.MoveParameters.Position >  axPositionLimits.PositionLimitPos THEN
    ax.MoveParameters.Position :=  axPositionLimits.PositionLimitPos;
  END_IF;
  IF ax.MoveParameters.Position <  axPositionLimits.PositionLimitNeg THEN
    ax.MoveParameters.Position :=  axPositionLimits.PositionLimitNeg;
  END_IF;

  // Velocity
  IF ax.MoveParameters.Velocity > ax.MoveParameters.VelocityMax THEN
    ax.MoveParameters.Velocity := ax.MoveParameters.VelocityMax;
  END_IF;
  IF ax.MoveParameters.Velocity < ax.MoveParameters.VelocityMin THEN
    ax.MoveParameters.Velocity := ax.MoveParameters.VelocityMin;
  END_IF;

  // Accel and decel
  IF ax.MoveParameters.Acceleration > ax.MoveParameters.AccelMax THEN
    ax.MoveParameters.Acceleration := ax.MoveParameters.AccelMax;
  END_IF;
  IF ax.MoveParameters.Acceleration < ax.MoveParameters.AccelMin THEN
    ax.MoveParameters.Acceleration := ax.MoveParameters.AccelMin;
  END_IF;

  IF ax.MoveParameters.Deceleration > ax.MoveParameters.DecelMax THEN
    ax.MoveParameters.Deceleration := ax.MoveParameters.DecelMax;
  END_IF;
  IF ax.MoveParameters.Deceleration < ax.MoveParameters.DecelMin THEN
    ax.MoveParameters.Deceleration := ax.MoveParameters.DecelMin;
  END_IF;

  // The execution behavior is determined by the inputs set elsewhere
  // in particular the sMot_AxisCommands XxxxCmd bits,
  // and the values in sMot_MoveParameters structure

  // Axis reference set in init routine

  // Only enable the fb if the axis is not set to be ignored
  // TODO: Different check needed? Not sure how to tell if an axis reference is not set
  // It would be nice to check ax.fbMpAxisBasic.MpLink <> 0 for example, but this is a structure not an address
  IF NOT ax.Ignore AND ax.AxisNo <> 0 THEN
    ax.fbMpAxisBasic.Enable := TRUE;
  ELSE
    ax.fbMpAxisBasic.Enable := FALSE;
  END_IF;

  // Load the parameters from the sMot_MoveParameter structure into
  // local structure variables used for the fb
  fctPackMpAxisBasicParams(_I_UdtParams:= ADR(ax.MoveParameters), _IO_MpParams := axisBasicParams);

  // To allow move parameter changes to take effect without having to stop,
  // detect a difference between the desired parameters and the previous values.
  // If they are different, then set the update bit until the UpdateDone bit is set.
  // NOTE: This fb manages the ax.fbMpAxisCoupling.Update request and monitors the .UpdateDone bit
  // Use the .UpdateCouplingParams bit in the command structure if the application needs to control
  // when to trigger the update. If parameters need to be set in possibly different areas of the software,
  // and all the updates should take place at once, the update fb is called conditionally. The
  // checked bit can be set high so it is called all the time if the checked bit is not managed.
  ax.Commands.UpdateMoveParams:= TRUE;
  IF ax.Commands.UpdateMoveParams THEN
    ax.fbUpdateBFbParams(_IO_MpParams := axisBasicParams);
    ax.Commands.UpdateMoveParams := FALSE;
  END_IF;

  // TODO: Enforce move permissives

  // Use the commands from the axis structue
  ax.fbMpAxisBasic.ErrorReset := ax.Commands.DriveResetCmd;
  ax.fbMpAxisBasic.Power := ax.Commands.EnableCmd;
  ax.fbMpAxisBasic.Home := ax.Commands.HomeCmd;
  // There is no specific jog cmd. Use Move Velocity instead.
  ax.fbMpAxisBasic.MoveVelocity := ax.Commands.MoveVelocityCmd OR ax.Commands.MoveJogCmd;
  ax.fbMpAxisBasic.MoveAbsolute := ax.Commands.MoveAbsoluteCmd;
  ax.fbMpAxisBasic.MoveAdditive := ax.Commands.MoveRelativeCmd;
  ax.fbMpAxisBasic.Stop := ax.Commands.StopCmd;
  ax.fbMpAxisBasic.JogPositive := ax.Commands.MoveJogPositiveCmd;
  ax.fbMpAxisBasic.JogNegative := ax.Commands.MoveJogNegativeCmd;
  ax.fbMpAxisBasic.LimitLoad := ax.MoveParameters.EnableTorqueLimit;
  ax.fbMpAxisBasic.ReleaseBrake := ax.Commands.ReleaseBrakeCmd;
  ax.fbMpAxisBasic.AutoTune := FALSE; // TODO
  ax.fbMpAxisBasic.Simulate := FALSE; // TODO

  // Call the fb
  ax.fbMpAxisBasic();

  // Update the axis status structure
  ax.Status.Position := ax.fbMpAxisBasic.Position;
  ax.Status.Velocity := ax.fbMpAxisBasic.Velocity;
  ax.Status.IsPoweredOn := ax.fbMpAxisBasic.PowerOn;
  ax.Status.IsHomed := ax.fbMpAxisBasic.IsHomed;
  ax.Status.IsInVelocity := ax.fbMpAxisBasic.InVelocity;
  ax.Status.IsInPosition := ax.fbMpAxisBasic.InPosition;
  ax.Status.IsMoveActive := ax.fbMpAxisBasic.MoveActive;
  ax.Status.IsMoveDone := ax.fbMpAxisBasic.MoveDone;
  ax.Status.IsStopped := ax.fbMpAxisBasic.Stopped;
  ax.Status.IsTorqueLimitReady := ax.fbMpAxisBasic.LimitLoadReady;
  ax.Status.IsBrakeManuallyReleased := ax.fbMpAxisBasic.BrakeReleased;

  // Now load the sMot_AxisStatus structure with the data returned from the fb
  fctGetMpAxisInfo(_I_MpInfo := ADR(ax.fbMpAxisBasic.Info), _IO_UdtStatus := ax.Status);

  // Calculate special (algorithmic) positions
  CalcSpecialPositions;

  // Now that the status of this axis is known, copy it to the other axes slave status
  // area if this axis is specified as a slave.
  CopySlaveStatusToMaster;

END_ACTION

ACTION ActionMpAxisCoupling:
  // 1) Packs the sMot_CouplingParameters into a local axisCouplingParamsStructure
  // 2) Detects parameter changes and manages the Update and UpdateDone bits
  // 3) Sets the fb command bits based on the axis sMot_AxisCommands structure
  // 4) Runs the fbMpAxisCoupling funciton block
  // 5) Updates the axis structure with the status and axis info coming back from the fb

  // The execution behavior is determined by the inputs set elsewhere
  // in particular the sMot_AxisCommands Engage/Disengage Slave bits,
  // and the values in sMot_CouplingParameters struture.

  // Axis references set in init routine

  // Only enable the coupling fb if the axis number has been set,
  // the slave axis number has been set, and neither is set to be ignored.
  IF NOT ax.Ignore AND ax.AxisNo <> AD_UNKNOWN AND
     ax.CouplingParameters.SlaveAxisNo <> AD_UNKNOWN AND
     NOT axes[ax.CouplingParameters.SlaveAxisNo].Ignore THEN
    ax.fbMpAxisCoupling.Enable := TRUE;
  ELSE
    ax.fbMpAxisCoupling.Enable := FALSE;
  END_IF;

  // If the slave axis has changed, update the fb link to the slave axis
  // Handle this change before the call to fbUpdateCFbParams because
  // a slave number change would be detected but not handled by fbUpdateCFbParams.
  IF ax.CouplingParameters.SlaveAxisNo <> ax.CouplingParametersPrev.SlaveAxisNo THEN
    // Set the axis object based on the slave number
    IF ax.CouplingParameters.SlaveAxisNo <> AD_UNKNOWN THEN
      ax.SlaveAxisObj := axes[ax.CouplingParameters.SlaveAxisNo].AxisObj;
    ELSE
      ax.SlaveAxisObj := axDummySlave;
    END_IF;
    ax.fbMpAxisCoupling.MpLink := ADR(ax.SlaveAxisObj);
    // Update the previous value now that the change is handled
    ax.CouplingParametersPrev.SlaveAxisNo := ax.CouplingParameters.SlaveAxisNo;
  END_IF;

  // Load the parameters from the sMot_CouplingParameters structure into
  // local structure variables used for the call to fbMpAxisCoupling
  fctPackMpAxisCouplingParams(_I_UdtParams:= ADR(ax.CouplingParameters), _IO_MpParams := axisCouplingParams);

  // To allow coupling parameter changes to take effect without having to stop,
  // detect a difference between the desired parameters and the previous values.
  // If they are different, then set the update bit until the UpdateDone bit is set.
  // NOTE: This fb manages the ax.fbMpAxisCoupling.Update request and monitors the .UpdateDone bit
  // Use the .UpdateCouplingParams bit in the command structure if the application needs to control
  // when to trigger the update. If parameters need to be set in possibly different areas of the software,
  // and all the updates should take place at once, the update fb is called conditionally. The
  // checked bit can be set high so it is called all the time if the checked bit is not managed.
  ax.Commands.UpdateCouplingParams:= TRUE;
  IF ax.CouplingParameters.SlaveAxisNo <> AD_UNKNOWN AND ax.Commands.UpdateCouplingParams THEN
    ax.fbUpdateCFbParams();
    ax.Commands.UpdateCouplingParams := FALSE;
  END_IF;

  // Use the commands from the axis structue
  ax.fbMpAxisCoupling.ErrorReset := ax.Commands.DriveResetCmd;

  // Gear in if there is a slave, it is requested and it is allowed by the slave
  ax.fbMpAxisCoupling.Gear := ax.CouplingParameters.SlaveAxisNo <> AD_UNKNOWN AND ax.CouplingParameters.GearInCmd AND axes[ax.CouplingParameters.SlaveAxisNo].CouplingParameters.CouplingPermissive;
  ax.fbMpAxisCoupling.Cam := FALSE; // Not using camming
  // Gear in position if there is a slave, it is requested and it is allowed by the slave
  ax.fbMpAxisCoupling.GearInPos := ax.CouplingParameters.SlaveAxisNo <> AD_UNKNOWN AND ax.CouplingParameters.GearInPosCmd AND axes[ax.CouplingParameters.SlaveAxisNo].CouplingParameters.CouplingPermissive;
  // Generate an offset or phase shift if there is a slave, it is requested and it is allowed by the slave
  ax.fbMpAxisCoupling.OffsetShift := ax.CouplingParameters.SlaveAxisNo <> AD_UNKNOWN AND ax.CouplingParameters.OffsetShiftCmd AND axes[ax.CouplingParameters.SlaveAxisNo].CouplingParameters.CouplingPermissive;
  ax.fbMpAxisCoupling.PhaseShift := ax.CouplingParameters.SlaveAxisNo <> AD_UNKNOWN AND ax.CouplingParameters.PhaseShiftCmd AND axes[ax.CouplingParameters.SlaveAxisNo].CouplingParameters.CouplingPermissive;
  ax.fbMpAxisCoupling.GetCamPosition := FALSE; // not using camming
  ax.fbMpAxisCoupling.CamPrepare := FALSE; // not using camming
  ax.fbMpAxisCoupling.Recovery := FALSE; // not using camming

  // Call the fb
  ax.fbMpAxisCoupling();

  // Update the axis status structure
  ax.Status.IsCoordInCompensation := ax.fbMpAxisCoupling.InCompensation;
  ax.Status.IsCoordInSync := ax.fbMpAxisCoupling.InSync;
  ax.Status.IsCoordOffsetDone := ax.fbMpAxisCoupling.OffsetDone;
  ax.Status.IsCoordPhasingDone := ax.fbMpAxisCoupling.PhasingDone;
  ax.Status.IsCoordRecoveryDone := ax.fbMpAxisCoupling.RecoveryDone;

  // Now load the sMot_AxisStatus structure with the data returned from the fb
  fctGetMpCouplingInfo(_I_MpInfo := ADR(ax.fbMpAxisCoupling.Info), _IO_UdtStatus := ax.Status);
  // add to the isCoordSlaveReady status the slave coupling permissive
  ax.Status.IsCoordSlaveReady := ax.Status.IsCoordSlaveReady AND axes[ax.CouplingParameters.SlaveAxisNo].CouplingParameters.CouplingPermissive;

END_ACTION

ACTION CalcSpecialPositions :
  // If there is an algorithm needed for calculating a different position, it can be done here
  // If not, just use the axis position.
  ax.Status.CalculatedPosition1 :=  ax.Status.Position;
  ax.Status.CalculatedPosition2 :=  ax.Status.Position;
  ax.Status.CalculatedPosition3 :=  ax.Status.Position;
END_ACTION

ACTION CopySlaveStatusToMaster :
  // If this axis number is a slave to another axis, then copy this axis
  // status to the master axis structure. This is a convenience
  // so the HMI for example, only needs to look in one structure (the master) and
  // can access the slave status.

  // Loop thru the axes. If the axis of index has this axis specified as a slave axis,
  // copy this axis status to the axis of index slave status.
  // Axis 0 is a dummy axis, so it can be skipped.
  FOR axIdx := 1 TO AXIS_COUNT DO
    IF axes[axIdx].CouplingParameters.SlaveAxisNo = AXIS_NO THEN
      // This axis is a slave to the axis referenced by axIdx.
      // Copy this axis status to the indexed axis slave status
      fctCopyAxisStatus(_I_SrcStatus := ADR(ax.Status), _I_DestStatus := ADR(axes[axIdx].StatusSlave));
    END_IF;
  END_FOR;
END_ACTION
```

- ActionMotionFbs.st.bak (not shown)
